{attribute addProperty BoxType "ELX9410-0000-0018"}
{attribute addProperty Id "UndervoltageAT %I*BOOL81"}
{attribute addProperty CRC "3645161568"}
{attribute addProperty SizeInBites "8"}
{attribute addProperty SizeInBytes "1"}
TYPE Status_Us_Out_D944C060 :
STRUCT
	{attribute addProperty Name "Undervoltage"}
	Undervoltage AT %I* : BOOL;
END_STRUCT
END_TYPE

(* stored: Version 1.2.0.0, ProductVersion 3.1.4024.9
   DUT Status_Us_Out_D944C060: Id {0907c031-cbd5-4ae9-8414-831622830728} *)
